// TIA Portal V18 export
TYPE "LGasp_typeListaPrd"
// stored: IsFailsafeCompliant false
   STRUCT
      prodfromPC : Array[1.."NumRigheProduzione"] of "LGasp_typeRigaProdfromPC";
      prodfromPLC : Array[1.."NumRigheProduzione"] of "LGasp_typeRigaProdfromPLC";
   END_STRUCT;
END_TYPE
